TYPE ST_HMI_MANUAL_DRIVE_OUT :
STRUCT
	bVisible			: BOOL;
	stObjectName		: ST_Text;
	stState				: ST_Text;
	stButtonJogPos,
	stButtonJogNeg,
	stButtonStop		: ST_HMI_BUTTON_OUT;
	aDriveModeName		: ARRAY[0..1] OF ST_Text;
END_STRUCT
END_TYPE

(* stored: Version 1.1.0.1, ProductVersion 3.1.4024.11
   DUT ST_HMI_MANUAL_DRIVE_OUT: Id {efc0debb-f797-4b15-960f-77b171310677} *)
